(* CoDeSys 2.3 export: CODETOTEXT.EXP *)

(* POU _FC/codeToText, ST *)
FUNCTION codeToText : STRING
VAR_INPUT
	input : WORD;
END_VAR
VAR
END_VAR
	CASE input OF
		0 : codeToText := 'Не готов';
		128 : codeToText := 'Готов';
		129 : codeToText := 'В работе';
		131 : codeToText := 'Разгон';
		133 : codeToText := 'Тормажение';
	ELSE
		RETURN;
	END_CASE;
END_FUNCTION
